PROGRAM _05_FLAGS
(****************************************************************************)
//FLAGS PROGRAMM
//	- Diverse Allgemeine Signale
//
//	04.09.2019/Dj
//
//	Version:
(****************************************************************************)
VAR_INPUT
	xIN_AIR			: 	BOOL;				//Luftdruck
	xIN_btRES_TEMP	:	structButton;		//BUTTON ResetCounter
END_VAR
VAR
	TOF_AirOFF		: 	TOF;				//Air NIO
	TON_btReset		:	TON;				//Reset Taste gedrückt
	
    _FB_Lampe		:   FB_LampeBNI007F;	//Lampe Balluf BN007F
	
	_FB_btRESET		: 	FB_BUTTON;			//Reset Temp Counter
	
END_VAR

//--------------------------------------------------------------------------
//Air ON
//--------------------------------------------------------------------------
TOF_AirOFF(IN:=xIN_AIR , PT:=T#500MS);
HMI.xAIRon	:= TOF_AirOFF.Q;

//--------------------------------------------------------------------------
//Reset Counter	
//--------------------------------------------------------------------------
//Button
_FB_btRESET(pbtIN:= ADR(xIN_btRES_TEMP),
	xINdis:= FALSE, 
	xINon:= (PERS.udiTempNOK=0) AND (PERS.udiTempOK=0), 
	xINerr:= FALSE);
TON_btReset(IN:=xIN_btRES_TEMP.press, PT:=T#1.5S);
//Reset
IF TON_btReset.Q THEN
	PERS.udiTempNOK:=0;
	PERS.udiTempOK:=0;
END_IF

//--------------------------------------------------------------------------
//Flanken
//--------------------------------------------------------------------------

END_PROGRAM

(* stored: Version 1.1.0.1, ProductVersion 3.1.4022.18
   POU _05_FLAGS: Id {55eeaa85-1eb4-4842-b105-d90f94beefba}, SpecialFunc None *)
